// TIA Portal V16 export
// export: Created 2024-09-05T17:36:33.9740354Z, ExportSetting WithDefaults, DisplayName Totally Integrated Automation Portal, DisplayVersion V16 Update 6, DisplayName TIA Portal Version Control Interface, DisplayVersion V16 Update 2, DisplayName TIA Portal Openness, DisplayVersion V16 Update 6, DisplayName STEP 7 Professional, DisplayVersion V16 Update 6, DisplayName STEP 7 Safety, DisplayVersion V16, DisplayName WinCC Advanced, DisplayVersion V16 Update 6
VAR_GLOBAL   // PLC tag table "_not used"
   SENSORES_LASER_OK AT %M2.3 : Bool;
   "1_OK" AT %M2.4 : Bool;
   RESET_MSG_INIT AT %M2.5 : Bool;
   M_TRC1_OK AT %M2.6 : Bool;
   M_TRC2_OK AT %M2.7 : Bool;
   M_TRC3_OK AT %M3.0 : Bool;
   M_TRC4_OK AT %M3.1 : Bool;
   M_PFC_OK AT %M3.2 : Bool;
   Prueba_Leyva AT %M3.3 : Bool;
END_VAR
